{attribute 'pack_mode' := '1'}
TYPE ST_3002_2_Manual_section EXTENDS ST_SectionHeader :
	STRUCT
		Enable_manual_control : E_3002_2_Enable_manual_control;
		Forward				  : E_3002_2_Inactive_Active;
		Backward			  : E_3002_2_Inactive_Active;
		Left				  : E_3002_2_Inactive_Active;
		Right				  : E_3002_2_Inactive_Active;
		Drive_speed			  : REAL; //The manual drive speed reference in meters per second.
	END_STRUCT
END_TYPE

(* stored: Version 1.1.0.1
   DUT ST_3002_2_Manual_section: Id {56dd65c4-740c-4d5d-9f05-3d6456820281} *)
